INTERFACE ILogger

METHOD Write : STRING
VAR_INPUT
	sMsg	: STRING;
END_VAR
END_METHOD

END_INTERFACE

(* stored: Version 1.1.0.1, ProductVersion 3.1.4024.12
   Itf ILogger: Id {1ce2a87c-b691-40d6-88e3-c310f1f514e4}
   Method Write: Id {86cda17a-eaf2-4088-b678-172c29ab6cd9} *)
